{attribute 'qualified_only'}
VAR_GLOBAL
	lamp : BOOL;
	knop : BOOL;
END_VAR

(* stored: Version 1.1.0.1, ProductVersion 3.1.4024.12
   GVL GVL: Id {73c2ae93-5fbd-4731-acda-a3b905b37dd3} *)
